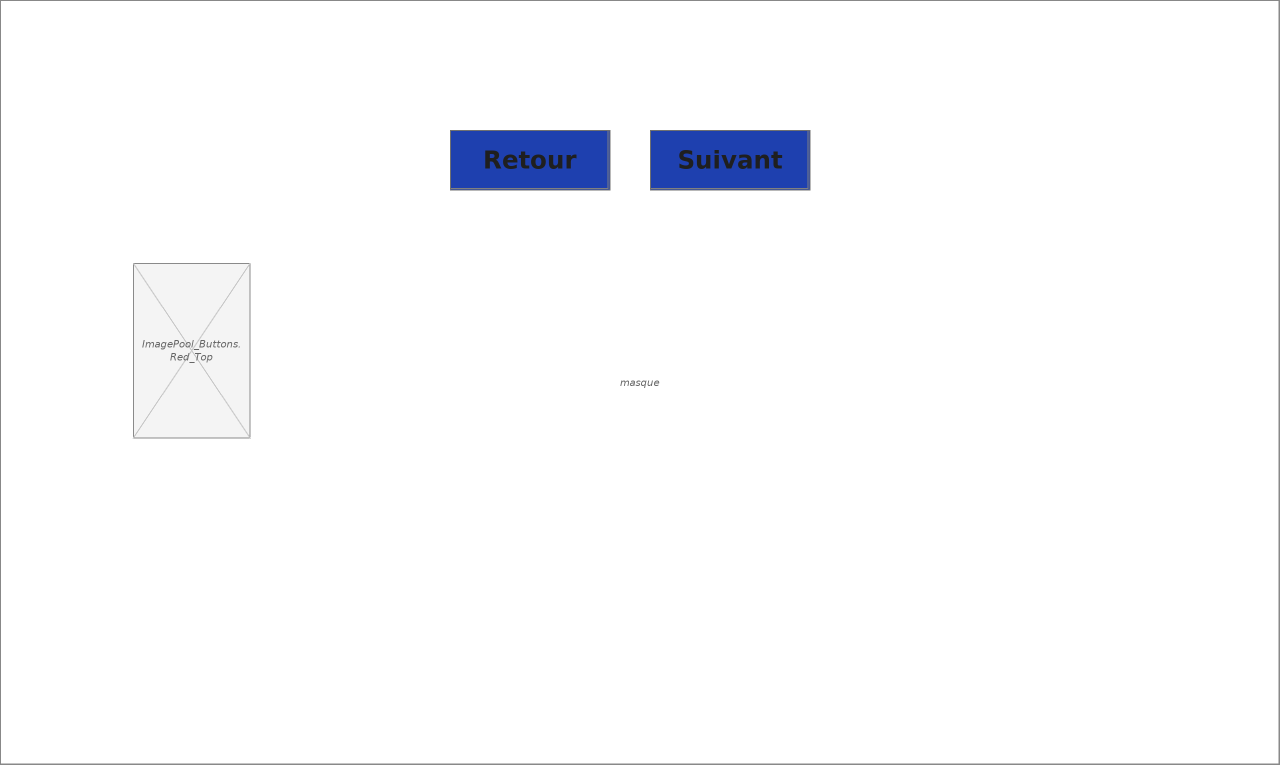
VISUALIZATION Maintenance_6  // 1280x765
    Frame (0,0 1280x765)
        shows masque()
    Button (650,130 160x60), "Suivant"
        OnMouseDown: change screen: Maintenance_7
    Button (450,130 160x60), "Retour"
        OnMouseDown: execute {
            IF (Option_Cabine_Climatique)
            	THEN
            	VisuElems.CURRENTVISU := 'Maintenance_5';
            	ELSIF (Option_WC_GV OR Option_WC_PV OR Option_Prise)
            		THEN
            		VisuElems.CURRENTVISU := 'Maintenance_4';
            	ELSIF (Option_Bas_Debit OR Option_Douchette OR Option_NEP)
            		THEN
            		VisuElems.CURRENTVISU := 'Maintenance_3';
            	ELSIF (Option_Douche OR Option_Lavabo)
            		THEN
            		VisuElems.CURRENTVISU := 'Maintenance_2';
            	ELSIF (Option_RegSouf_Ultrason OR Option_Reg_Etanche_Ext OR Option_V3V_EauMitig)
            		THEN
            		VisuElems.CURRENTVISU := 'Maintenance_1';
            	ELSE
            	VisuElems.CURRENTVISU := 'menu';
            END_IF
        }
    Group (64,209 463x544), invisible if: NOT Option_Com_RegSouf_Ultrason
        Rectangle (0,0 463x64), "COM Registre soufflage"
        Group (69,54 326x175)
            Group (0,0 117x175)
                Image (0,0 117x175), invisible if: Enable_ecr_param_Reg_Souf, image: ImagePool_Buttons.Green_Bottom
                    OnMouseDown: toggle Enable_ecr_param_Reg_Souf
                Image (0,0 117x175), invisible if: NOT Enable_ecr_param_Reg_Souf, image: ImagePool_Buttons.Red_Top
                    OnMouseDown: toggle Enable_ecr_param_Reg_Souf
            Rectangle (114,64 212x48), "Ecr paramètres"
        RoundedRectangle (32,225 398x64), "Debit Max : %d Vol/h", text variable: Ecriture_Cons_Max_Reg_Souf
            OnMouseDown: write the text variable via VisuDialogs.Numpad, min 0, max 1000, format %d
        Rectangle (32,353 398x64), "Debit Max : %d Vol/h", text variable: Lecture_Cons_Max_Reg_Souf
        Rectangle (32,416 398x64), "Debit Min : %d Vol/h", text variable: Lecture_Cons_Min_Reg_Souf
        RoundedRectangle (32,289 398x64), "Debit Min : %d Vol/h", text variable: Ecriture_Cons_Min_Reg_Souf
            OnMouseDown: write the text variable via VisuDialogs.Numpad, min 0, max 1000, format %d
        Rectangle (32,480 398x64), "Position : %.0f %%", text variable: MES_Pos_Reg_Souf
END_VISUALIZATION

(* stored: Version 1.1.0.1, ProductVersion 3.1.4024.16
   Visu Maintenance_6: Id {7497dcdd-7005-487d-a797-1db8166d9233} *)
